// TIA Portal V20 export
VAR_GLOBAL   // PLC tag table "SR-X100W_Entrace"
   Entrace_Read_Complete AT %I700.0 : Bool;
   Entrace_Read_Failure AT %I701.0 : Bool;
   Entrace_Read_Data AT %I702.0 : "SR-X100W_Read_Data";
   Entrace_Read_Request AT %Q700.0 : Bool;
   Entrace_Read_Complete_Clear AT %Q701.0 : Bool;
END_VAR
